FUNCTION wr_state_v : BOOL
VAR_INPUT
	state : INT;
END_VAR
VAR
END_VAR

wr_state_v := FALSE;
//WRITE FLAGS STATE-MACHINE #################(PLC->VISION SYSTEM)
Vision_struct.States.Val1:=state;
Vision_struct.States.Val2:=state;
Vision_struct.States.Val3:=state;
wr_state_v := TRUE;

END_FUNCTION

(* stored: Version 1.1.0.1, ProductVersion 3.1.4024.4
   POU wr_state_v: Id {a566cb6c-9f01-43fe-80a0-d336ca04a601}, SpecialFunc None *)
